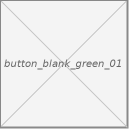
VISUALIZATION Green_Ind  // 129x129
VAR_INPUT
	m_Input_Inst : Bool;
END_VAR
    Image (0,0 127x127), invisible if: (m_Input_Inst) <> 0, image: button_blank_gray_01
    Image (0,0 127x127), invisible if: (NOT m_Input_Inst) <> 0, image: button_blank_green_01
END_VISUALIZATION

(* stored: Version 1.1.0.1, ProductVersion 3.1.4018.2
   Visu Green_Ind: Id {bc370c22-626c-41d6-9e84-1471601440a9} *)
